FUNCTION_BLOCK State_CMD_ATV320 (* Basic Function Block Type *)
  (* Standard: 61499-2 *)
  (* Version 0.0, 05/08/2021, SESA371406, Schneider Electric, Template *)
  PACKAGE SE.Nereda;
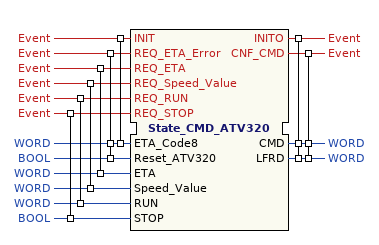
  EVENT_INPUT
    INIT WITH ETA_Code8; (* Initialization Request *)
    REQ_ETA_Error WITH Reset_ATV320, ETA_Code8; (* Normal Execution Request *)
    REQ_ETA WITH ETA;
    REQ_Speed_Value WITH Speed_Value;
    REQ_RUN WITH RUN;
    REQ_STOP WITH STOP;
  END_EVENT
  EVENT_OUTPUT
    INITO WITH CMD, LFRD; (* Initialization Confirm *)
    CNF_CMD WITH CMD, LFRD;
  END_EVENT
  VAR_INPUT
    ETA_Code8 : WORD; (* Input event qualifier *)
    Reset_ATV320 : BOOL;
    ETA : WORD;
    Speed_Value : WORD;
    RUN : WORD;
    STOP : BOOL;
  END_VAR
  VAR_OUTPUT
    CMD : WORD; (* Output event qualifier *)
    LFRD : WORD;
  END_VAR
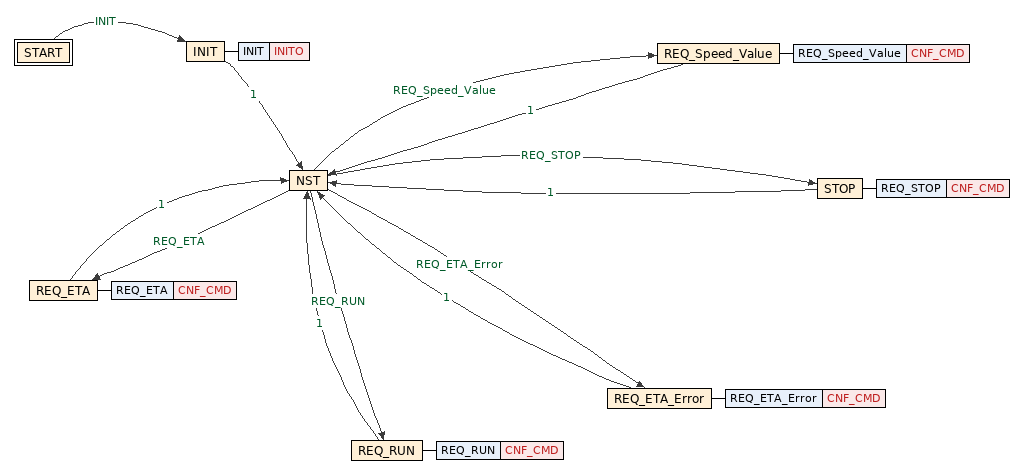
  EC_STATES
    START; (* Initial State *)
    INIT : INIT -> INITO; (* Initialization *)
    REQ_ETA_Error : REQ_ETA_Error -> CNF_CMD; (* Normal execution *)
    REQ_ETA : REQ_ETA -> CNF_CMD;
    NST;
    REQ_Speed_Value : REQ_Speed_Value -> CNF_CMD;
    REQ_RUN : REQ_RUN -> CNF_CMD;
    STOP : REQ_STOP -> CNF_CMD;
  END_STATES
  EC_TRANSITIONS
    START TO INIT := INIT;
    REQ_ETA TO NST := 1;
    INIT TO NST := 1;
    NST TO REQ_ETA := REQ_ETA;
    NST TO REQ_ETA_Error := REQ_ETA_Error;
    REQ_ETA_Error TO NST := 1;
    NST TO REQ_Speed_Value := REQ_Speed_Value;
    REQ_Speed_Value TO NST := 1;
    REQ_RUN TO NST := 1;
    NST TO REQ_RUN := REQ_RUN;
    STOP TO NST := 1;
    NST TO STOP := REQ_STOP;
  END_TRANSITIONS
  ALGORITHM INIT IN ST: (* Initialization algorithm *)
;

	CMD := 16#80;
  END_ALGORITHM
  ALGORITHM REQ_ETA_Error IN ST: (* Normally executed algorithm *)
;

(*IF Reset_ATV320 =TRUE THEN
	CMD := 16#80;
END_IF;*)

IF ETA_Code8 = 16#8 AND Reset_ATV320 =TRUE THEN
	CMD := 16#80;
	Reset_ATV320 := FALSE;
END_IF;
  END_ALGORITHM
  ALGORITHM REQ_ETA IN ST:
;

IF ETA = 16#50  THEN
	CMD := 16#6;
END_IF;

IF ETA = 16#31  THEN
	CMD := 16#7;
END_IF;
  END_ALGORITHM
  ALGORITHM REQ_Speed_Value IN ST:
;

LFRD:=Speed_Value;
  END_ALGORITHM
  ALGORITHM REQ_RUN IN ST:
;

IF RUN = 16#F AND ETA = 16#33 AND STOP = FALSE THEN
	CMD:= 16#F;
END_IF;

IF RUN = 16#7 AND ETA = 16#37 THEN
	CMD:= 16#7;
END_IF;
  END_ALGORITHM
  ALGORITHM REQ_STOP IN ST:
;

IF STOP = TRUE AND (CMD = 16#F OR CMD =16#7) THEN
	CMD:= 16#2;
END_IF;

IF STOP = FALSE AND ETA = 16#17 THEN
	CMD:= 16#0;
END_IF;
  END_ALGORITHM
END_FUNCTION_BLOCK
